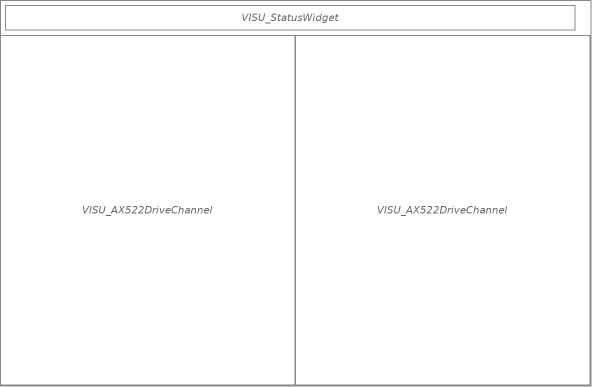
VISUALIZATION VISU_AX522Drive  // 592x387
VAR_IN_OUT
    ref : AX52XXDrive;
    widget : AX52XXDriveWidget;
END_VAR
    Frame (5,5 570x25)
        shows VISU_StatusWidget(widget := widget.actualStatus)
    Frame (0,35 295x350)
        shows VISU_AX522DriveChannel(ref := ref.parts.channelA, widget := widget.channelA)
    Frame (295,35 295x350)
        shows VISU_AX522DriveChannel(ref := ref.parts.channelB, widget := widget.channelB)
END_VISUALIZATION

(* stored: Version 1.1.0.1, ProductVersion 3.1.4019.2
   Visu VISU_AX522Drive: Id {e9b50dc5-8a90-4d0a-b55c-3b020a3a2d79} *)
